# EPICS substitutions: jawsManagerApp/Db/jaws_manager_test.substitutions
global {P=\$(P), SAMPLE_JAW=SAMPLE, MOD_TO_SAMPLE=100, MOD_WIDTH=20, MOD_HEIGHT=10}

file "$(TOP)/jawsManagerApp/Db/common.template" {
	{DIR=H}
	{DIR=V}
}

file "$(TOP)/jawsManagerApp/Db/jaws_manager_single.template" {
    { JAW="JAWS1", MOD_TO_JAW="20"}
    { JAW="JAWS2", MOD_TO_JAW="50"}
}
